FUNCTION_BLOCK FB_Stepper EXTENDS FB_Device
VAR_INPUT	
END_VAR
VAR_OUTPUT
END_VAR
VAR
END_VAR

//Add the tc2_mc function blocks here

END_FUNCTION_BLOCK

(* stored: Version 1.1.0.1
   POU FB_Stepper: Id {a38730a4-3247-47f2-8174-116774cc335c}, SpecialFunc None *)
